FUNCTION_BLOCK FB_FeedCircle EXTENDS FB_RecipeBase

METHOD Build : BOOL
VAR
    TotalX, Radius : LREAL;
    Velo : LREAL;
    localConfig : ST_GantryXYZ_Config;
    LeadInY : LREAL := 20.0;
    LeadOutY : LREAL := 20.0;
END_VAR
_Busy := TRUE;
_Done := FALSE;
_Error := FALSE;
Build := FALSE;

THIS^.UpdateNestingLimits();

IF NOT _Config.IsValid THEN
    _Busy := FALSE;
    _Error := TRUE;
    RETURN;
END_IF

TotalX := _Config.Diameter;
Radius := TotalX / 2.0;

// ===================================================
// DEFINICJA ILOŚCI I PUNKTÓW STARTOWYCH
// ===================================================
_ShapesCount := 1; 

_ShapeStart[1].X := TotalX;
_ShapeStart[1].Y := Radius - LeadInY;

IF _ConfigProvider <> 0 THEN
    localConfig := _ConfigProvider.Config;
    Velo := localConfig.CuttingSpeedXY;
ELSE
    Velo := 50.0;
END_IF

_GeometryWriter.Clear();
_GeometryWriter.EnableTangentialFollowing();

// RYSOWANIE TYLKO TEGO KSZTAŁTU, O KTÓRY PROSI EXECUTOR
CASE _CurrentShapeIndex OF
    1:
        _GeometryWriter.AddStartPoint(_ShapeStart[1].X, _ShapeStart[1].Y); 
        _GeometryWriter.AddLine(TotalX, Radius, Velo); 
        _GeometryWriter.AddArc(0.0, Radius, Radius, Radius, Velo, FALSE);
        _GeometryWriter.AddArc(TotalX, Radius, Radius, Radius, Velo, FALSE);
        _GeometryWriter.AddLine(TotalX, Radius + LeadOutY, Velo); 
END_CASE

_GeometryWriter.EndTable();

_Busy := FALSE;
_Done := TRUE;
Build := TRUE;
END_METHOD

METHOD PROTECTED CalculateFootprint
VAR_INPUT
END_VAR
_NominalX := _Config.Diameter;
_NominalY := _Config.Diameter;
END_METHOD

PROPERTY ExecutionRoute : E_ExecutionRoute
GET
ExecutionRoute := E_ExecutionRoute.eFeedTable;
END_GET
END_PROPERTY

METHOD FB_init : BOOL
VAR_INPUT
	bInitRetains : BOOL; // if TRUE, the retain variables are initialized (warm start / cold start)
	bInCopyCode : BOOL;  // if TRUE, the instance afterwards gets moved into the copy code (online change)
END_VAR
_Limits.Diameter.MinVal := 50.0;
_Limits.Diameter.MaxVal := 1200.0;
_Limits.Radius.MinVal := 10.0;
_Limits.Radius.MaxVal := 100;

_Limits.CuttingOverpass.MinVal := 0.0;
_Limits.CuttingOverpass.MaxVal := 50.0;
_Limits.GroovingOverpass.MinVal := 0.0;
_Limits.GroovingOverpass.MaxVal := 50.0;
END_METHOD

END_FUNCTION_BLOCK

(* stored: Version 1.1.0.1, ProductVersion 3.1.4024.15
   POU FB_FeedCircle: Id {e9adcfe5-7e4a-4852-a853-8210a47fd80c}, SpecialFunc None
   Method Build: Id {cd170bea-55d1-4b18-9d93-4857d1144680}
   Method CalculateFootprint: Id {bcba16d7-1bb9-45ef-95d7-88011fb53b8e}
   Property ExecutionRoute: Id {d2087356-9a9c-4c33-89d5-bf6c71c7e6ae}
   Get Get: Id {7fbe3751-e710-423a-8f1b-b2644f0b3a95}
   Method FB_init: Id {3462e180-3698-449a-9577-fb4640fc1cef} *)
